VAR_GLOBAL CONSTANT
	ATM	:	REAL := 760; // Atmospheric pressure in Torr
	tSec : INT := 1; // time in seconds
	IonMassRate : REAL := 0.00001; // Torr*Liter/seconds
END_VAR

(* stored: Version 1.1.0.1, ProductVersion 3.1.4020.12
   GVL GVL_VSS_CONSTANT: Id {ae843ad2-19d5-47c3-859e-73fc00707dcb} *)
